FUNCTION FC_SET_BIT_IN_BYTE : BOOL
VAR_INPUT
	Value : BOOL;
	RefByte : POINTER TO BYTE;
	BitToSet : USINT;
END_VAR
VAR
END_VAR

CASE BitToSet OF
	
	0:
		RefByte^.0 := Value;
	1:
		RefByte^.1 := Value;
	2:
		RefByte^.2 := Value;
	3:
		RefByte^.3 := Value;
	4:
		RefByte^.4 := Value;
	5:
		RefByte^.5 := Value;
	6:	
		RefByte^.6 := Value;
	7:
		RefByte^.7 := Value;
		
END_CASE;

END_FUNCTION

(* stored: Version 1.1.0.1, ProductVersion 3.1.4024.12
   POU FC_SET_BIT_IN_BYTE: Id {fa8b4505-2d40-4dab-b30f-a7ff7c6c8df0}, SpecialFunc None *)
